(* PLC project Unnamed, Unknown Unnamed 1 *)
(* stored: creationDateTime 2024-12-16T21:18:47, modificationDateTime 2024-12-16T23:14:50 *)

PROGRAM Stoplight
  VAR
    COUNTER : DINT;
    STOPLIGHT_TIME : DINT := 100;
    TIMER : BOOL;
    A1 : BOOL;
    A2 : BOOL;
    AP : BOOL;
    B1 : BOOL;
    B2 : BOOL;
    BP : BOOL;
    C1 : BOOL;
    C2 : BOOL;
    CP : BOOL;
  END_VAR
  VAR  (* added by the conversion: wires and edge detectors of the diagram *)
    _MOVE47_ENO : BOOL;
    _MOVE47_OUT : DINT;
    _EQ39_OUT : BOOL;
    _EQ41_OUT : BOOL;
    _EQ43_OUT : BOOL;
  END_VAR

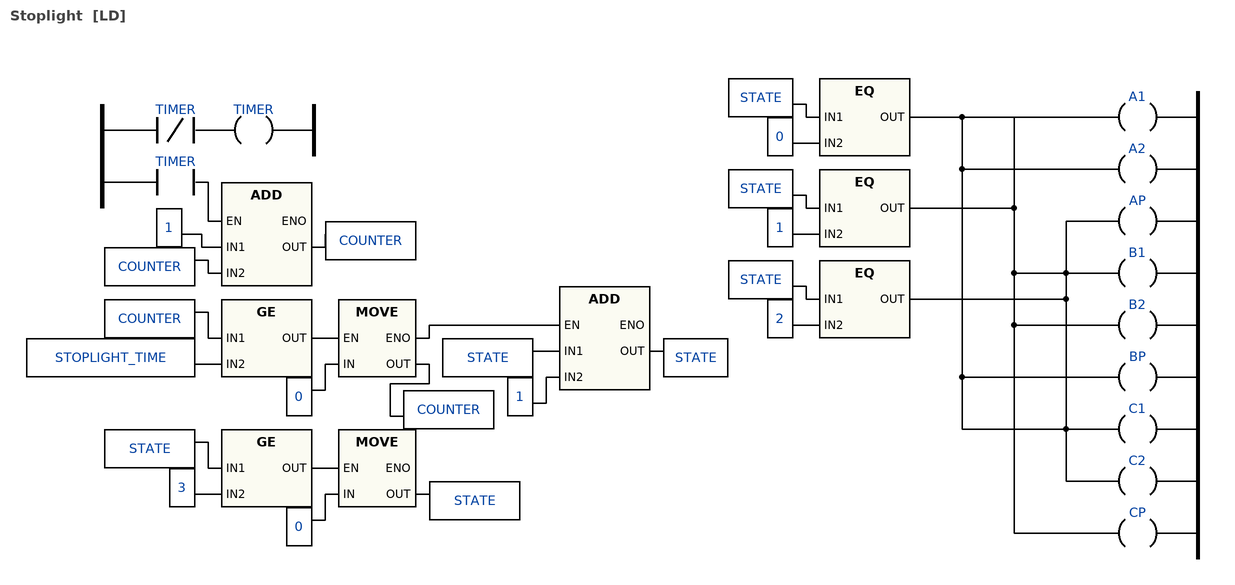
(* LD diagram, written out as Structured Text *)
TIMER := NOT TIMER;
IF TIMER THEN COUNTER := 1 + COUNTER; END_IF;
_MOVE47_OUT := MOVE(EN := COUNTER >= STOPLIGHT_TIME, IN := 0, ENO => _MOVE47_ENO);
IF _MOVE47_ENO THEN COUNTER := _MOVE47_OUT; END_IF;
IF _MOVE47_ENO THEN STATE := STATE + 1; END_IF;
IF STATE >= 3 THEN STATE := 0; END_IF;
_EQ39_OUT := STATE = 0;
_EQ41_OUT := STATE = 1;
A1 := _EQ39_OUT OR _EQ41_OUT;
A2 := _EQ39_OUT;
_EQ43_OUT := STATE = 2;
AP := _EQ43_OUT;
B1 := _EQ41_OUT OR _EQ43_OUT;
B2 := _EQ41_OUT;
BP := _EQ39_OUT;
C2 := _EQ43_OUT;
C1 := _EQ43_OUT OR _EQ39_OUT;
CP := _EQ41_OUT;
END_PROGRAM

CONFIGURATION Config0
  RESOURCE Res0 ON PLC
    TASK task0(INTERVAL := T#20ms, PRIORITY := 0);
    PROGRAM instance0 WITH task0 : Stoplight;
  END_RESOURCE
END_CONFIGURATION
